FUNCTION FLogging : BOOL
VAR_INPUT

///SDOC/////////////////////////////////////////////////////////////////////////
//
//  FLogging.TcPOU      - Function - PLC state logging - AVT PLC 
//
//  Author:         Mark Colvin                         Date: Sept 5, 2018
//
//	Beckhoff TC3 Structured Text for CX8190 PLC
//
//	includes features:
//		10 inker enables
///////////////////////////////////////////////////////////////////////SDOCEND//
//inputs to this function

	b_enabled :BOOL;	//enabled - enable or disable logging
	w_state	:WORD;	//state to be logged
END_VAR
VAR

	w_count		:WORD;	//temp
	w_max_count	:WORD;	//temp
END_VAR

(************************************************************************************************
 *
 *   FUNCTION 	:FLogging
 *
 *   Author		:	Mark Colvin
 *
 *   Description:	Write logging of states for system log text file 'tcsyslog' in My Device folder of PLC; ADSLOG_MSGTYPE_LOG
 *				(or the IDE output window; ADSLOG_MSGTYPE_HINT)
 *
 *   Parameters	:	enabled - enable or disable logging
 *					state to be logged
 *
 *   Returns	:	void	
 *
 *   History	:   13-Sep-18	MarkC	Created
 *
************************************************************************************************)
w_max_count := 10000;  // this count does not seem to work, control logging externally with logging enable

if((b_enabled = TRUE) AND (w_count < w_max_count)) THEN
	ADSLOGDINT( msgCtrlMask := ADSLOG_MSGTYPE_LOG OR ADSLOG_MSGTYPE_HINT, msgFmtStr := 'Sweep Value state: %d', dintArg:=  w_state);
	w_count := w_count +1;
END_IF 
if( b_enabled = FALSE) THEN
	w_count := 0;
END_IF

FLogging:= FALSE;

RETURN;

END_FUNCTION

(* stored: Version 1.1.0.1, ProductVersion 3.1.4022.6
   POU FLogging: Id {d7bd57ae-2c0e-4ed7-a69b-3257f3f83fbb}, SpecialFunc None *)
